FUNCTION_BLOCK ModelBA (* Composite Function Block Type *)
  (* Standard: 61499-2 *)
  (* Version 0.2, 2003-12-05, JHC, Rockwell Automation, Renamed from NEWCOMPFB. *)
  (* Version 0.1, 2002-01-08, JHC, Rockwell Automation, Added DLY FB as example. *)
  (* Version 0.0, 2000-05-27, JHC, Rockwell Automation *)
  (* Compiler header: package fb.rt.pnp; *)
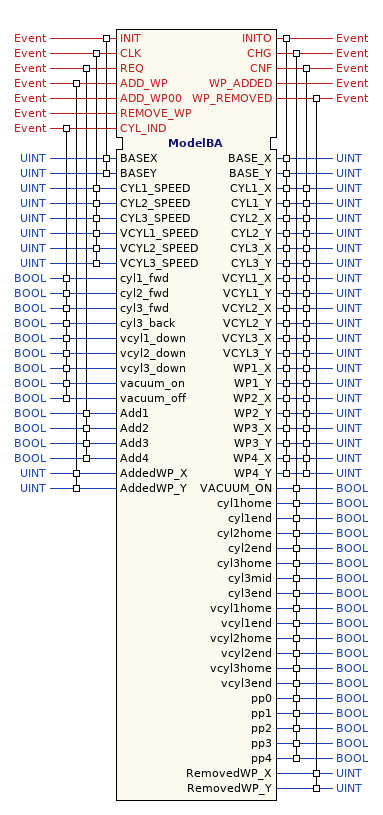
  EVENT_INPUT
    INIT WITH BASEX, BASEY; (* Initialization Request *)
    CLK WITH CYL1_SPEED, CYL2_SPEED, VCYL1_SPEED, CYL3_SPEED, VCYL2_SPEED, VCYL3_SPEED; (* Clock *)
    REQ WITH Add1, Add2, Add3, Add4;
    ADD_WP WITH AddedWP_X, AddedWP_Y;
    ADD_WP00;
    REMOVE_WP;
    CYL_IND WITH cyl1_fwd, cyl2_fwd, vcyl1_down, vacuum_on, vacuum_off, cyl3_fwd, cyl3_back, vcyl2_down, vcyl3_down;
  END_EVENT
  EVENT_OUTPUT
    INITO WITH BASE_X, BASE_Y, CYL1_Y, CYL2_Y, CYL1_X, CYL2_X, CYL3_Y, CYL3_X, VCYL1_X, VCYL1_Y, VCYL2_X, VCYL2_Y, VCYL3_X, VCYL3_Y, WP1_X, WP1_Y, WP2_X, WP2_Y, WP3_X, WP3_Y, WP4_X, WP4_Y; (* Initialization Confirm *)
    CHG WITH pp0, pp1, pp2, pp3, pp4, VACUUM_ON, cyl1home, cyl1end, cyl2home, cyl2end, cyl3home, cyl3end, vcyl1home, vcyl1end, vcyl2home, vcyl2end, vcyl3home, vcyl3end, cyl3mid; (* View State Changed *)
    CNF WITH VCYL1_Y, WP1_X, WP1_Y, WP2_X, WP2_Y, WP3_X, WP3_Y, WP4_X, WP4_Y, CYL2_X, VCYL1_X, CYL2_Y, CYL1_Y, CYL1_X, CYL3_Y, CYL3_X, VCYL2_X, VCYL2_Y, VCYL3_X, VCYL3_Y;
    WP_ADDED;
    WP_REMOVED WITH RemovedWP_X, RemovedWP_Y;
  END_EVENT
  VAR_INPUT
    BASEX : UINT;
    BASEY : UINT;
    CYL1_SPEED : UINT;
    CYL2_SPEED : UINT;
    CYL3_SPEED : UINT;
    VCYL1_SPEED : UINT;
    VCYL2_SPEED : UINT;
    VCYL3_SPEED : UINT;
    cyl1_fwd : BOOL;
    cyl2_fwd : BOOL;
    cyl3_fwd : BOOL;
    cyl3_back : BOOL;
    vcyl1_down : BOOL;
    vcyl2_down : BOOL;
    vcyl3_down : BOOL;
    vacuum_on : BOOL;
    vacuum_off : BOOL;
    Add1 : BOOL;
    Add2 : BOOL;
    Add3 : BOOL;
    Add4 : BOOL;
    AddedWP_X : UINT;
    AddedWP_Y : UINT;
  END_VAR
  VAR_OUTPUT
    BASE_X : UINT; (* Response Data from Socket *)
    BASE_Y : UINT; (* Response Data from Socket *)
    CYL1_X : UINT; (* Response Data from Socket *)
    CYL1_Y : UINT; (* Response Data from Socket *)
    CYL2_X : UINT; (* Response Data from Socket *)
    CYL2_Y : UINT; (* Response Data from Socket *)
    CYL3_X : UINT; (* Response Data from Socket *)
    CYL3_Y : UINT; (* Response Data from Socket *)
    VCYL1_X : UINT; (* Response Data from Socket *)
    VCYL1_Y : UINT; (* Response Data from Socket *)
    VCYL2_X : UINT; (* Response Data from Socket *)
    VCYL2_Y : UINT; (* Response Data from Socket *)
    VCYL3_X : UINT; (* Response Data from Socket *)
    VCYL3_Y : UINT; (* Response Data from Socket *)
    WP1_X : UINT; (* Response Data from Socket *)
    WP1_Y : UINT; (* Response Data from Socket *)
    WP2_X : UINT; (* Response Data from Socket *)
    WP2_Y : UINT; (* Response Data from Socket *)
    WP3_X : UINT; (* Response Data from Socket *)
    WP3_Y : UINT; (* Response Data from Socket *)
    WP4_X : UINT; (* Response Data from Socket *)
    WP4_Y : UINT; (* Response Data from Socket *)
    VACUUM_ON : BOOL; (* Response Data from Socket *)
    cyl1home : BOOL;
    cyl1end : BOOL;
    cyl2home : BOOL;
    cyl2end : BOOL;
    cyl3home : BOOL;
    cyl3mid : BOOL;
    cyl3end : BOOL;
    vcyl1home : BOOL;
    vcyl1end : BOOL;
    vcyl2home : BOOL;
    vcyl2end : BOOL;
    vcyl3home : BOOL;
    vcyl3end : BOOL;
    pp0 : BOOL;
    pp1 : BOOL;
    pp2 : BOOL;
    pp3 : BOOL;
    pp4 : BOOL;
    RemovedWP_X : UINT;
    RemovedWP_Y : UINT;
  END_VAR
  FBS
    Cylinder : PnpCylindersBA(InitialPosition := 0.0, HomeSensorRange := [0,1], MidSensorRange := [49,51], EndSensorRange := [99,100], Loaded := 0, LoadType := 0, CYL1MovingtDistance := 75, CYL2MovingtDistance := 75, CYL3MovingtDistance := 150, VCYL1MovingtDistance := 75, VCYL2MovingtDistance := 75, VCYL3MovingtDistance := 75);
    ViewControl : PnpXYCalculatorBA;
    SuctionUnit : PnPVacuum;
    WPSensors : WPsensorBA;
  END_FBS
  EVENT_CONNECTIONS
    INIT TO Cylinder.INIT;
    REQ TO ViewControl.REQ;
    ADD_WP TO ViewControl.ADD_WP;
    ADD_WP00 TO ViewControl.ADD_WP00;
    REMOVE_WP TO ViewControl.REMOVE_WP;
    ViewControl.WP_ADDED TO WP_ADDED;
    ViewControl.WP_REMOVED TO WP_REMOVED;
    Cylinder.INITO TO SuctionUnit.INIT;
    SuctionUnit.INITO TO ViewControl.INIT;
    CLK TO Cylinder.CLK;
    CYL_IND TO Cylinder.CYL_IND;
    CYL_IND TO SuctionUnit.CLK;
    SuctionUnit.CHG TO ViewControl.CLK;
    ViewControl.INITO TO WPSensors.INIT;
    WPSensors.CNF TO CHG;
    WPSensors.INITO TO INITO;
    ViewControl.CNF TO WPSensors.REQ;
    Cylinder.CNF TO ViewControl.CLK;
    Cylinder.CHG TO CHG;
    SuctionUnit.CHG TO CHG;
    ViewControl.CNF TO CNF;
  END_CONNECTIONS
  DATA_CONNECTIONS
    ViewControl.BASE_X TO BASE_X;
    ViewControl.BASE_Y TO BASE_Y;
    ViewControl.CYL1_X TO CYL1_X;
    ViewControl.CYL1_Y TO CYL1_Y;
    ViewControl.CYL2_X TO CYL2_X;
    ViewControl.CYL2_Y TO CYL2_Y;
    ViewControl.VCYL1_X TO VCYL1_X;
    ViewControl.VCYL1_Y TO VCYL1_Y;
    ViewControl.WP1_X TO WP1_X;
    ViewControl.WP1_Y TO WP1_Y;
    ViewControl.WP2_X TO WP2_X;
    ViewControl.WP2_Y TO WP2_Y;
    ViewControl.WP3_X TO WP3_X;
    ViewControl.WP3_Y TO WP3_Y;
    BASEX TO ViewControl.BASEX;
    BASEY TO ViewControl.BASEY;
    vacuum_on TO ViewControl.vacuum_on;
    vacuum_off TO ViewControl.vacuum_off;
    Add1 TO ViewControl.Add1;
    Add2 TO ViewControl.Add2;
    Add3 TO ViewControl.Add3;
    AddedWP_X TO ViewControl.AddedWP_X;
    AddedWP_Y TO ViewControl.AddedWP_Y;
    SuctionUnit.VacState TO VACUUM_ON;
    vacuum_on TO SuctionUnit.VacuumOn;
    vacuum_off TO SuctionUnit.VacuumOff;
    SuctionUnit.VacState TO ViewControl.vacuumon;
    ViewControl.WP1_X TO WPSensors.WP1_X;
    ViewControl.WP1_Y TO WPSensors.WP1_Y;
    ViewControl.WP2_X TO WPSensors.WP2_X;
    ViewControl.WP2_Y TO WPSensors.WP2_Y;
    ViewControl.WP3_X TO WPSensors.WP3_X;
    ViewControl.WP3_Y TO WPSensors.WP3_Y;
    WPSensors.wp11 TO pp0;
    WPSensors.wp14 TO pp3;
    WPSensors.wp13 TO pp2;
    WPSensors.wp12 TO pp1;
    cyl1_fwd TO Cylinder.CYL1Extend;
    CYL1_SPEED TO Cylinder.CYL1ForwardSpeed;
    CYL2_SPEED TO Cylinder.CYL2BackwardSpeed;
    CYL2_SPEED TO Cylinder.CYL2ForwardSpeed;
    CYL1_SPEED TO Cylinder.CYL1BackwardSpeed;
    cyl2_fwd TO Cylinder.CYL2Extend;
    cyl3_fwd TO Cylinder.CYL3Extend;
    cyl3_back TO Cylinder.CYL3Retract;
    CYL3_SPEED TO Cylinder.CYL3ForwardSpeed;
    CYL3_SPEED TO Cylinder.CYL3BackwardSpeed;
    vcyl1_down TO Cylinder.VCYL1Extend;
    VCYL1_SPEED TO Cylinder.VCYL1ForwardSpeed;
    VCYL1_SPEED TO Cylinder.VCYL1BackwardSpeed;
    vcyl2_down TO Cylinder.VCYL2Extend;
    VCYL2_SPEED TO Cylinder.VCYL2ForwardSpeed;
    VCYL2_SPEED TO Cylinder.VCYL2BackwardSpeed;
    vcyl3_down TO Cylinder.VCYL3Extend;
    VCYL3_SPEED TO Cylinder.VCYL3ForwardSpeed;
    VCYL3_SPEED TO Cylinder.VCYL3BackwardSpeed;
    WPSensors.wp15 TO pp4;
    ViewControl.CYL3_X TO CYL3_X;
    ViewControl.CYL3_Y TO CYL3_Y;
    ViewControl.VCYL2_X TO VCYL2_X;
    ViewControl.VCYL2_Y TO VCYL2_Y;
    ViewControl.VCYL3_X TO VCYL3_X;
    ViewControl.VCYL3_Y TO VCYL3_Y;
    Cylinder.CYL1AbsolutePos TO ViewControl.CYL1Pos;
    Cylinder.CYL2AbsolutePos TO ViewControl.CYL2Pos;
    Cylinder.CYL3AbsolutePos TO ViewControl.CYL3Pos;
    Cylinder.VCYL1AbsolutePos TO ViewControl.VCYL1Pos;
    Cylinder.VCYL2AbsolutePos TO ViewControl.VCYL2Pos;
    Cylinder.VCYL3AbsolutePos TO ViewControl.VCYL3Pos;
    Add4 TO ViewControl.Add4;
    Cylinder.CYL1AtHome TO cyl1home;
    Cylinder.CYL1AtEnd TO cyl1end;
    Cylinder.CYL2AtHome TO cyl2home;
    Cylinder.CYL2AtEnd TO cyl2end;
    Cylinder.CYL3AtHome TO cyl3home;
    Cylinder.CYL3AtEnd TO cyl3end;
    Cylinder.VCYL1AtHome TO vcyl1home;
    Cylinder.VCYL1AtEnd TO vcyl1end;
    Cylinder.VCYL2AtHome TO vcyl2home;
    Cylinder.VCYL2AtEnd TO vcyl2end;
    Cylinder.VCYL3AtHome TO vcyl3home;
    Cylinder.VCYL3AtEnd TO vcyl3end;
    Cylinder.CYL3AtMid TO cyl3mid;
  END_CONNECTIONS
END_FUNCTION_BLOCK
